// TwinCAT 3 PLC project MQTT
// ProgramVersion: 3.1.4023.0
// libraries:
//   Tc2_DataExchange, * (Beckhoff Automation GmbH)
//   Tc2_Standard, * (Beckhoff Automation GmbH)
//   Tc2_System, * (Beckhoff Automation GmbH)
//   Tc2_Utilities, * (Beckhoff Automation GmbH)
//   Tc3_Database, * (Beckhoff Automation GmbH)
//   Tc3_IotBase, * (Beckhoff Automation GmbH)
//   Tc3_Module, * (Beckhoff Automation GmbH)
// project tree:
//   DUTs/ WindTurbineData.TcDUT, E_DbLogState.TcDUT, STDBData.TcDUT
//   GVLs/ GVL_MQTT_Common.TcGVL, GVL_MQTT_Conf.TcGVL, GVL_ShellyRecentValues.TcGVL
//   / PlcTask.TcTTO
//   POUs/ MAIN.TcPOU, P_ADSCommManager.TcPOU, P_DatabaseExchange.TcPOU, P_MQTT_Agent.TcPOU
// real-time tasks:
//   TASK PlcTask: cycle T#10ms, priority 20, ADS port 350

CONFIGURATION MQTT
    RESOURCE PLC ON TwinCAT3
        TASK PlcTask(INTERVAL := T#10ms, PRIORITY := 20);
        PROGRAM MAIN WITH PlcTask : MAIN;
    END_RESOURCE
END_CONFIGURATION

// ---- DUTs/WindTurbineData.TcDUT
TYPE WindTurbineData :
STRUCT
    
    {attribute 'TagName' := 'ID'}
    WindTurbineID : STRING(255);
    
    {attribute 'FieldName' := 'Power'}
    Power : LREAL := -1; // ]
    
    {attribute 'FieldName' := 'Wind Speed'}
    WindSpeed : LREAL := -1; // [0) [m/s]
    
    {attribute 'FieldName' := 'Wind Direction'}
    WindDirection : LREAL := -1; // [0,360][°]
    
END_STRUCT
END_TYPE

// ---- DUTs/E_DbLogState.TcDUT
{attribute 'qualified_only'}
{attribute 'strict'}
TYPE E_DbLogState :
(
    idle := 0,
    init,
    writing,
    error
);
END_TYPE

// ---- DUTs/STDBData.TcDUT
TYPE STDBData :
STRUCT
    {attribute 'TagName' := 'ID'}
	sShellyID		:	STRING(255);
	
    {attribute 'FieldName' := 'Temperature'}
	rTemperature	:	LREAL;
	
    {attribute 'FieldName' := 'Humidity'}
	rHumidity		:	LREAL;
	
    {attribute 'FieldName' := 'Power'}
	iBatteryLevel	:	LINT;
	
END_STRUCT
END_TYPE

// ---- GVLs/GVL_MQTT_Common.TcGVL
{attribute 'qualified_only'}
VAR_GLOBAL
	bRestartServer	: BOOL;
	bNewDataJustCame : BOOL;
END_VAR

// ---- GVLs/GVL_MQTT_Conf.TcGVL
{attribute 'qualified_only'}
VAR_GLOBAL
	sServerIp			:	STRING := '10.24.102.185';
	sServerPort			:	UINT  := 1883;
	bServerError		:	BOOL;
	hrErrCode			:	HRESULT;
	bErr				:	BOOL;
	bConnected			:	BOOL;
	
	sMainTopic			:	STRING	:= 'shellies'	;
	sDevice				:	STRING	:=	'shellyht-1E7CD0';
	sSubTopic			:	STRING;
	
	sTempTopic			:	STRING := '/sensor/temperature';
	sHumTopic			:	STRING := '/sensor/humidity';
	sBatTopic			:	STRING := '/sensor/battery';
	sTimeStamp			:	STRING;
	sFullTempTopic		:	STRING ;
	sFullHumTopic		:	STRING ;
	sFullBatTopic		:	STRING ;
	
	
END_VAR

// ---- GVLs/GVL_ShellyRecentValues.TcGVL
{attribute 'qualified_only'}
VAR_GLOBAL
	rTemperature	:	REAL;
	rHumidity		:	REAL;
	iBatteryLevel	:	INT;
END_VAR

// ---- POUs/MAIN.TcPOU
PROGRAM MAIN
VAR
	bDoOnce : bool := true;
END_VAR

IF bDoOnce THEN
	bDoOnce := FALSE;
	P_ADSCommManager.FB_init(FALSE,FALSE);
END_IF
P_MQTT_Agent();
P_DatabaseExchange();
//P_DBTest();
P_ADSCommManager();

END_PROGRAM

// ---- POUs/P_ADSCommManager.TcPOU
PROGRAM P_ADSCommManager
VAR // comm values
	bValueToWrite		:	BOOL;
	bAutoWriteNewVal	:	BOOL;
	bWriteNewValOnce	:	BOOL;
	bCurrentValue		:	BOOL;
	sVarName			:	STRING(255) := 'P_Kuchnia._fbHeater_0.bManualValveOpen';
END_VAR
VAR
	fbWrite				:	FB_WriteAdsSymByName;
	fbRead				:	FB_ReadAdsSymByName;
	fbRTrigWriteOnce	:	R_TRIG;
	fbTonAutoWrite		:	TON := (pt := T#1S);
	iSwitch				:	INT := 1;
	bWriteInProgress	:	BOOL;
END_VAR

fbRTrigWriteOnce(clk := bWriteNewValOnce);
fbTonAutoWrite(IN := NOT fbTonAutoWrite.Q);
IF bAutoWriteNewVal OR fbread.bBusy THEN
	CASE iSwitch OF 
		1:
			IF fbTonAutoWrite.Q THEN
				fbRead(bRead := TRUE,
					sVarName := sVarName,
					nDestAddr := ADR(bCurrentValue),
					nLen := SIZEOF(bcurrentValue));
			END_IF
			fbRead();
			IF NOT fbRead.bBusy	AND NOT fbRead.bError THEN
				fbRead(bRead := FALSE);
				iSwitch := 2;
			END_IF
		2:
			IF bCurrentValue <> bValueToWrite THEN
				fbWrite(bWrite := TRUE,
					sVarName := sVarName,
					nSrcAddr := ADR(bValueToWrite),
					nlen := SIZEOF(bValueToWrite));
				IF NOT fbWrite.bBusy AND  NOT fbWrite.bError THEN
					fbWrite(bWrite := FALSE);
					iSwitch := 1;
				END_IF
			END_IF
	END_CASE
END_IF
IF fbRTrigWriteOnce.Q OR bWriteInProgress THEN
	fbWrite(bWrite := TRUE,
					sVarName := sVarName,
					nSrcAddr := ADR(bValueToWrite),
					nlen := SIZEOF(bValueToWrite));
	bWriteInProgress := TRUE;
	IF NOT fbWrite.bBusy AND  NOT fbWrite.bError THEN
		fbRead(bRead := TRUE,
			sVarName := sVarName,
			nDestAddr := ADR(bCurrentValue),
			nLen := SIZEOF(bcurrentValue));
		IF NOT fbRead.bBusy	AND NOT fbRead.bError THEN
			fbRead(bRead := FALSE);
			fbWrite(bWrite := FALSE);
			bWriteInProgress := FALSE;
		END_IF
	END_IF
END_IF

METHOD FB_init : BOOL
VAR_INPUT
	bInitRetains : BOOL := FALSE; // if TRUE, the retain variables are initialized (warm start / cold start)
	bInCopyCode : BOOL := FALSE;  // if TRUE, the instance afterwards gets moved into the copy code (online change)
END_VAR
fbRead.eComMode := E_AdsComMode.eAdsComModeFastCom;
fbRead.sNetId := '5.21.22.214.1.1';
fbRead.nPort := 851;
fbWrite.eComMode := E_AdsComMode.eAdsComModeFastCom;
fbWrite.sNetId := '5.21.22.214.1.1';
fbWrite.nPort := 851;
END_METHOD

END_PROGRAM

// ---- POUs/P_MQTT_Agent.TcPOU
PROGRAM P_MQTT_Agent
VAR
	fbIoTManager			:	FB_IotMqttClient;
    fbMessageQueue 			: 	FB_IotMqttMessageQueue;
    fbMessage      			: 	FB_IotMqttMessage;
    fbGetSystemTime         : GETSYSTEMTIME;
    fileTime        		: T_FILETIME;
	
	bTopicsSubscribed		:	BOOL;
	bConfigured				:	BOOL;
	sBuffer					:	STRING;
END_VAR

IF NOT bConfigured THEN 
	bConfigured := TRUE;
	
	fbIoTManager.sHostName  := GVL_MQTT_Conf.sServerIp;
	fbIoTManager.nHostPort	:= GVL_MQTT_Conf.sServerPort;
	fbIoTManager.sTopicPrefix := CONCAT(STR1 := GVL_MQTT_Conf.sMainTopic,str2 := 
												concat(str1 := '/',STR2 := GVL_MQTT_Conf.sDevice));
	fbIoTManager.ipMessageQueue	:=	fbMessageQueue;
ELSE
	fbIoTManager.Execute(bConnect := TRUE);
END_IF


IF fbIoTManager.bConnected AND NOT bTopicsSubscribed THEN 
	M_SubscribeToTopics();
END_IF

IF fbMessageQueue.nQueuedMessages <> 0 THEN 
	fbMessageQueue.Dequeue(fbMessage := fbMessage);
	
	IF fbMessage.CompareTopic(sTopic := GVL_MQTT_Conf.sFullBatTopic) THEN
		fbMessage.GetPayload(pPayload := ADR(sBuffer),
							nPayloadSize := fbMessage.nPayloadSize,
							bSetNullTermination := FALSE);
		GVL_ShellyRecentValues.iBatteryLevel := STRING_TO_INT(sBuffer);
	ELSIF fbMessage.CompareTopic(sTopic := GVL_MQTT_Conf.sFullHumTopic) THEN
		fbMessage.GetPayload(pPayload := ADR(sBuffer),
							nPayloadSize := fbMessage.nPayloadSize,
							bSetNullTermination := FALSE);
		GVL_ShellyRecentValues.rHumidity := STRING_TO_REAL(sBuffer);
	ELSIF fbMessage.CompareTopic(sTopic := GVL_MQTT_Conf.sFullTempTopic) THEN
		fbMessage.GetPayload(pPayload := ADR(sBuffer),
							nPayloadSize := fbMessage.nPayloadSize,
							bSetNullTermination := FALSE);
		GVL_ShellyRecentValues.rTemperature := STRING_TO_REAL(sBuffer);
	END_IF
	
	IF fbMessageQueue.nQueuedMessages  = 0 THEN 
		fbGetSystemTime(timeLoDW=>fileTime.dwLowDateTime, timeHiDW=>fileTime.dwHighDateTime );
		GVL_MQTT_Conf.sTimeStamp :=SYSTEMTIME_TO_STRING( FILETIME_TO_SYSTEMTIME( fileTime ) );
		GVL_MQTT_Common.bNewDataJustCame := TRUE;
	END_IF
	
END_IF








IF GVL_MQTT_Common.bRestartServer THEN
	M_NewConf();
	GVL_MQTT_Common.bRestartServer := FALSE;
	M_UnsubscribeToTopics();
END_IF
GVL_MQTT_Conf.bConnected	:=	fbIoTManager.bConnected;
GVL_MQTT_Conf.bErr			:=	fbIoTManager.bError;
GVL_MQTT_Conf.hrErrCode		:=	fbIoTManager.hrErrorCode;

METHOD M_NewConf : BOOL
VAR_INPUT
END_VAR
bConfigured := FALSE;
fbIoTManager.Execute(bConnect := false);
END_METHOD

METHOD M_SubscribeToTopics : BOOL
VAR_INPUT
END_VAR
IF 		fbIoTManager.Subscribe(sTopic := GVL_MQTT_Conf.sHumTopic,eQoS := TcIotMqttQos.ExactlyOnceDelivery)AND
	fbIoTManager.Subscribe(sTopic := GVL_MQTT_Conf.sTempTopic,eQoS := TcIotMqttQos.ExactlyOnceDelivery)AND
	fbIoTManager.Subscribe(sTopic := GVL_MQTT_Conf.sBatTopic,eQoS := TcIotMqttQos.ExactlyOnceDelivery) THEN
	M_SubscribeToTopics := FALSE;
	bTopicsSubscribed := TRUE;
	GVL_MQTT_Conf.sFullBatTopic := CONCAT(STR1 := fbIoTManager.sTopicPrefix,STR2:= GVL_MQTT_Conf.sBatTopic);
	GVL_MQTT_Conf.sFullHumTopic := CONCAT(STR1 := fbIoTManager.sTopicPrefix,STR2:= GVL_MQTT_Conf.sHumTopic);
	GVL_MQTT_Conf.sFullTempTopic := CONCAT(STR1 := fbIoTManager.sTopicPrefix,STR2:= GVL_MQTT_Conf.sTempTopic);
ELSE
	M_SubscribeToTopics := TRUE;
END_IF
END_METHOD

METHOD M_UnsubscribeToTopics : BOOL
VAR_INPUT
END_VAR
IF 	fbIoTManager.Unsubscribe(sTopic := GVL_MQTT_Conf.sHumTopic)AND
	fbIoTManager.Unsubscribe(sTopic := GVL_MQTT_Conf.sTempTopic)AND
	fbIoTManager.Unsubscribe(sTopic := GVL_MQTT_Conf.sBatTopic) THEN
	M_UnsubscribeToTopics := FALSE;
	bTopicsSubscribed := FALSE;
ELSE
	M_UnsubscribeToTopics := TRUE;
END_IF
END_METHOD

END_PROGRAM

// ---- POUs/P_DatabaseExchange.TcPOU
PROGRAM P_DatabaseExchange
VAR
	State									: E_DbLogState;
    QueryOption_TSDB_Insert 				: T_QueryOptionTimeSeriesDB_Insert; // defines detailed Queryparameter
    fbNoSQLQueryBuilder_TimeSeriesDB 		: FB_NoSQLQueryBuilder_TimeSeriesDB; // defines database type specific api
    fbNoSqlQueryEvt 						: FB_NoSQLQueryEvt(sNetID := '', tTimeout := T#15S); // functionblock to execute queries
    
    // error handling helper values
    TcResult								: Tc3_Database.I_TcMessage;
	
    bError									: BOOL;
    bWriting								: BOOL; // Set this bool fla to write the data once into the InfluxDB
    udiDatabaseID							: UDINT := 1; // Handle to the configured database
    sErrorMessage							: STRING(255);
	
	stDbData								: STDBData;
	fbPlowToDatabase						: TON := (PT := t#10s);
END_VAR

fbPlowToDatabase(in := NOT fbPlowToDatabase.Q);
CASE State OF 
	E_DbLogState.idle:
		 IF GVL_MQTT_Common.bNewDataJustCame OR fbPlowToDatabase.Q THEN
			 GVL_MQTT_Common.bNewDataJustCame := FALSE;
			 state := E_DbLogState.init;
		 END_IF
	E_DbLogState.init:
		fbNoSQLQueryBuilder_TimeSeriesDB.pQueryOptions := ADR(QueryOption_TSDB_Insert);
        fbNoSQLQueryBuilder_TimeSeriesDB.cbQueryOptions := SIZEOF(QueryOption_TSDB_Insert);    
        stDbData.iBatteryLevel := GVL_ShellyRecentValues.iBatteryLevel;
		stDbData.rHumidity		:= GVL_ShellyRecentValues.rHumidity;
		stDbData.rTemperature	:= GVL_ShellyRecentValues.rTemperature;
		stDbData.sShellyID		:= GVL_MQTT_Conf.sDevice;
        QueryOption_TSDB_Insert.sTableName := 'ShellyTemperature';
        QueryOption_TSDB_Insert.sDataType := 'STDBData';
        QueryOption_TSDB_Insert.pSymbol := ADR(stDbData);
        QueryOption_TSDB_Insert.cbSymbol := SIZEOF(stDbData);
        QueryOption_TSDB_Insert.nDataCount := 1;
        QueryOption_TSDB_Insert.nStartTimestamp := F_GetSystemTime();
        QueryOption_TSDB_Insert.nCycleTime := 10000; // (in 100 ns)
        State := E_DbLogState.writing;
		bError := FALSE;
		sErrorMessage :='OK';
	E_DbLogState.writing:
        IF fbNoSqlQueryEvt.Execute(udiDatabaseID, fbNoSQLQueryBuilder_TimeSeriesDB) THEN
            IF fbNoSqlQueryEvt.bError THEN
                TcResult := fbNoSqlQueryEvt.ipTcResult;                
                State := E_DbLogState.error;
            ELSE
                State := E_DbLogState.idle;
            END_IF
        END_IF
	
	E_DbLogState.error:
        
        IF TcResult.RequestEventText(1033, sErrorMessage, SIZEOF(sErrorMessage)) THEN
            TcResult.Send(F_GetSystemTime());
            State := E_DbLogState.idle;
            bError := TRUE;
        END_IF
	
END_CASE

END_PROGRAM
